// TIA Portal V20 export
TYPE "UDT_typeMeasureInput"
   STRUCT
      input : Struct
         bo_Active : Bool;
         mode : Int;
      END_STRUCT;
      output : Struct
         done : Bool;
         busy : Bool;
         error : Bool;
         i32_ErrorCode : Word;
         r64_MeasuredValue1 : LReal;
         r64_MeasuredValue2 : LReal;
      END_STRUCT;
   END_STRUCT;
END_TYPE
